{attribute addProperty BoxType "EL2034-0000-0016"}
{attribute addProperty Id "DiagAT %I*ARRAY[0..3] OF Diag_4CD4E3A23240ChannelAT %Q*ARRAY[0..3] OF Channel_7F374EB03240WcStateAT %I*WcState_98A4DF7520.250InfoDataAT %I*InfoData_192954DE1620"}
{attribute addProperty CRC "3400452497"}
{attribute addProperty SizeInBites "82"}
{attribute addProperty SizeInBytes "10.25"}
TYPE EL2034_14D53AA6 :
STRUCT
	{attribute addProperty Name "Diag"}
	Diag : ARRAY[0..3] OF Diag_4CD4E3A2;
	{attribute addProperty Name "Channel"}
	Channel : ARRAY[0..3] OF Channel_7F374EB0;
	{attribute addProperty Name "WcState"}
	WcState : WcState_98A4DF75;
	{attribute addProperty Name "InfoData"}
	InfoData : InfoData_192954DE;
END_STRUCT
END_TYPE

(* stored: Version 1.2.0.0, ProductVersion 3.1.4024.9
   DUT EL2034_14D53AA6: Id {6ae92a9f-1b41-4310-b84f-eb7f6ddb4ec2} *)
